// Interlock logic for the Amphos shutter
FUNCTION F_AmphosShutterEnable : BOOL
VAR_INPUT
	bAmphosOn : BOOL; // Whether the amphos is on
	fOpcpaVoltage : LREAL; // The voltage of the OPCPA
	bLoopTempOverride01 : BOOL; // Whether the chiller loop error is overriden
	bLoopTempOverride02 : BOOL; // Whether the chiller loop error is overriden
	bLoopTempOverride03 : BOOL; // Whether the chiller loop error is overriden
	bLoopTempOverride04 : BOOL; // Whether the chiller loop error is overriden
	bMasterOverride : BOOL; //Master manual override control input
	bAmpShutterClosed : BOOL; //Master Amphos shutter control. TRUE = Closed
END_VAR
VAR_IN_OUT CONSTANT
	stErrors : ST_ErrorStates; // Currently detected errors
	stOpcpaSetpoints : ST_LaserSetpoints; // OPCPA setpoints
END_VAR
VAR
END_VAR

IF (stErrors.bHardwareFailure // Close shutter if there is a hardware failure
	OR stErrors.bLeakOpticalTableAmphosOn OR stErrors.bLeakOpcpaCarbideOn (* OR stErrors.bLeakUnderTable *) // Close shutter if there is a leak on the optical table with the amphos on, a leak under the table, or a leak inside the OPCPA with Carbide on
	OR bAmphosOn AND (
		(NOT bLoopTempOverride01 AND stErrors.bChillerLoop01) OR 
		(NOT bLoopTempOverride02 AND stErrors.bChillerLoop02) OR 
		(NOT bLoopTempOverride03 AND stErrors.bChillerLoop03) OR 
		(NOT bLoopTempOverride04 AND stErrors.bChillerLoop04)) // Close shutter if the amphos is on and the temperature is too high in any loop. Ignore if operator override is enabled
	OR (stErrors.bOpcpaBeam) // Close shutter if in OPCPA beam error state and OPCPA voltage too low
	(*OR stErrors.bTempMon01 OR stErrors.bTempMon02 OR stErrors.bTempMon03 OR stErrors.bTempMon04 OR stErrors.bTempMon05 OR 
		stErrors.bTempMon06 OR stErrors.bTempMon07 OR stErrors.bTempMon08 // Close shutter if temperature too high at any monitor location *)
	OR stErrors.bDumpChiller) // Close shutter if there is a Dump Chiller error
	(* OR stErrors.bAmphosMRC02 OR stErrors.bAmphosMRC03 // Close shutter if there are errors on the additional MRCs *)
	AND NOT bMasterOverride //if master override is TRUE, ignore all errors
THEN
	F_AmphosShutterEnable := FALSE;
ELSIF bMasterOverride AND bAmpShutterClosed THEN
	F_AmphosShutterEnable := FALSE;
ELSIF bMasterOverride AND NOT bAmpShutterClosed THEN
	F_AmphosShutterEnable := TRUE;
ELSE
	F_AmphosShutterEnable := TRUE;
END_IF

END_FUNCTION

(* stored: Version 1.1.0.1, ProductVersion 3.1.4024.6
   POU F_AmphosShutterEnable: Id {a786de1e-4080-488b-a915-5c3ae196891d}, SpecialFunc None *)
